// TIA Portal project "test2" (V17)

(* hardware
DEVICE "S7-1200 station_1"  S7-1200 Station
   slot 0: "Rack_0"  S7-1200 Rack  Rack  V1.0
   slot 1: "PLC_1"  CPU 1214C DC/DC/DC  6ES7 214-1AG40-0XB0  V4.3
*)

// ===== PLC "PLC_1"  CPU 1214C DC/DC/DC =====

VAR_GLOBAL   // PLC tag table "Default tag table"
   "sensor" AT %I0.0 : Bool;
   "bangtai" AT %Q0.1 : Bool;
   "start_xla" AT %M10.0 : Bool;
   "delay5s" AT %M10.2 : Bool;
   "Tag_1" AT %M50.0 : Bool;
   "Tag_2" AT %M60.0 : Bool;
END_VAR

DATA_BLOCK "DB1"   // DB1
{ S7_Optimized_Access := 'FALSE' }
VERSION : 0.1
   VAR
      data : Word;
   END_VAR
BEGIN
END_DATA_BLOCK

DATA_BLOCK "DB3"   // DB3
{ S7_Optimized_Access := 'FALSE' }
VERSION : 0.1
   VAR
      Start_Xla : Int;
   END_VAR
BEGIN
END_DATA_BLOCK

// folder: System blocks/Program resources

DATA_BLOCK "TON1"   // DB2
{ S7_Optimized_Access := 'TRUE' }
AUTHOR : Simatic
FAMILY : IEC
NAME : IEC_TMR
VERSION : 1.0
// stored: InstanceOfName IEC_TIMER
"IEC_TIMER"
BEGIN
END_DATA_BLOCK

DATA_BLOCK "TON4"   // DB5
{ S7_Optimized_Access := 'TRUE' }
AUTHOR : Simatic
FAMILY : IEC
NAME : IEC_TMR
VERSION : 1.0
// stored: InstanceOfName IEC_TIMER
"IEC_TIMER"
BEGIN
END_DATA_BLOCK

// folder: (top level)

ORGANIZATION_BLOCK "Main"   // OB1, LAD, ProgramCycle
TITLE = "Main Program Sweep (Cycle)"
{ S7_Optimized_Access := 'TRUE' }
VERSION : 0.1
   VAR_INPUT
      Initial_Call : Bool;   // Initial call of this OB
      Remanence : Bool;   // =True, if remanent data are available
   END_VAR
   VAR_TEMP   // added for the SCL form of the ladder/FBD networks
      _w1 : Bool;
   END_VAR
BEGIN

REGION Network 1: chay bang tai
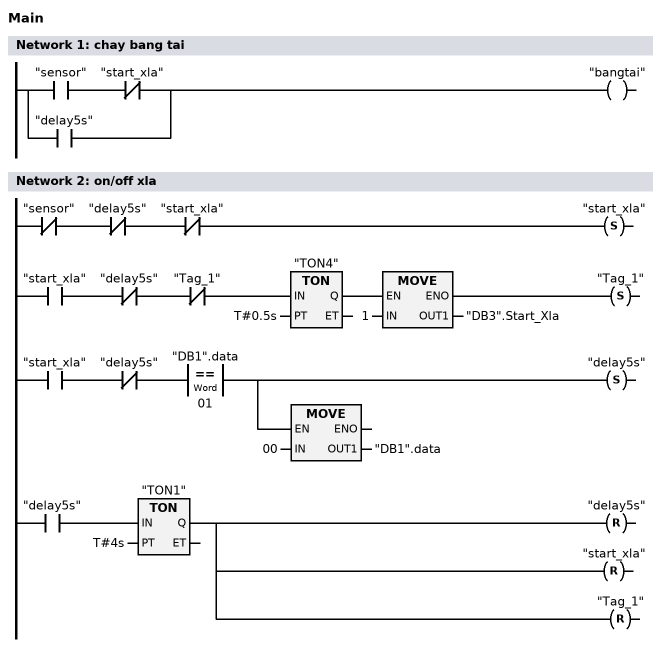
   RUNG wire#powerrail
      Contact( "sensor" )
      I_Contact( "start_xla" )
      wire#w1
      Coil( "bangtai" )
   END_RUNG
   RUNG wire#powerrail
      Contact( "delay5s" )
   END_RUNG wire#w1
   // the same network as SCL:
   "bangtai" := ("sensor" AND NOT "start_xla") OR "delay5s";
END_REGION

REGION Network 2: on/off xla
   IF NOT "sensor" AND NOT "delay5s" AND NOT "start_xla" THEN "start_xla" := TRUE; END_IF;
   "TON4".TON(IN := "start_xla" AND NOT "delay5s" AND NOT "Tag_1", PT := T#0.5s);
   IF "TON4".Q THEN
       "DB3".Start_Xla := 1;
       "Tag_1" := TRUE;
   END_IF;
   #_w1 := "start_xla" AND NOT "delay5s" AND ("DB1".data = 01);
   IF #_w1 THEN
       "delay5s" := TRUE;
       "DB1".data := 00;
   END_IF;
   "TON1".TON(IN := "delay5s", PT := T#4s);
   IF "TON1".Q THEN
       "delay5s" := FALSE;
       "start_xla" := FALSE;
       "Tag_1" := FALSE;
   END_IF;
END_REGION
END_ORGANIZATION_BLOCK